{attribute 'qualified_only'}
TYPE E_PML_Command :
(
    None := 0,
    Reset,
    Start,
    Stop,
    Pause,    // maps to Hold/Held path
    Resume,   // maps to Unholding->Execute
    Abort
) := None;
END_TYPE

(* stored: Version 1.1.0.1, ProductVersion 3.1.4024.13
   DUT E_PML_Command: Id {69cc6e69-4fff-44a2-8bc6-87073577c8be} *)
